FUNCTION_BLOCK CM_SpeedDoor EXTENDS CM_Base IMPLEMENTS I_Door
VAR_INPUT
	i_stSettings : ST_SettingsSpeedDoor;
END_VAR
VAR
	// Inputs
	I_bStaDoorIsOpended AT %I* : BOOL; //Door is opened
	I_bStaDoorIsClosed AT %I* : BOOL; //Door is closed
	I_bStaDoorHasError AT %I* : BOOL; //Door has error
	
	// Outputs
	Q_bCmdOpenDoor AT %Q* : BOOL; //Commnad to open door
	Q_bCmdCloseDoor AT %Q* : BOOL; //Command to close door
	Q_bCmdResetDoor AT %Q* : BOOL; //Command to reset door (controller)
		
	// Requests
	s_bReqClose : BOOL;
	s_bReqOpen : BOOL;
	s_bReqReset : BOOL;
	
	// States
	s_bStaDoorIsClosed : BOOL;
	s_bStaDoorIsClosing : BOOL;
	s_bStaDoorIsOpened : BOOL;
	s_bStaDoorIsOpening : BOOL;
	s_bStaDoorHasError : BOOL;
	
	// Timers
	s_tofResetPulse : TOF;
	s_tonTimeput : TON;
	
	
	// Feedbacks
	arr_sFeedbackName : ARRAY[0..7] OF STRING;
	arr_bFeedbackState : ARRAY[0..7] OF STRING;
	
	
	// Alarms
	s_errSpeedDoor : FB_AlarmHandler;
	s_errTimeout : FB_AlarmHandler;
		
END_VAR


SUPER^();

METHOD PROTECTED _m_Alarms : BOOL
VAR
	nCounter : UDINT;
	
	tTimeout : TIME;
	sMessage : STRING(8);
END_VAR

IF NOT SUPER^._m_Alarms() THEN
	RETURN;
END_IF

s_errSpeedDoor(
	i_bStaActive := i_bReqEnable AND s_bStaDoorHasError, 
	i_eAlarmLevel := E_AlarmLevel.Alarm,
	i_sAlarmText := CONCAT(i_sCmName , CONCAT(': Drive/Controller - ', 'has error (check DYNACO-system)'))
);

IF s_bReqOpen THEN
	tTimeout := i_stSettings.tDoorOpeningTimeout;
	sMessage := 'opening';
ELSIF s_bReqClose THEN
	tTimeout := i_stSettings.tDoorClosingTimeout;
	sMessage :=	'closing';
ELSE
	tTimeout := T#60S;
	sMessage :=	'unknown';	
END_IF
 
s_tonTimeput(
	IN := (s_bReqOpen AND NOT s_bStaDoorIsOpened) OR (s_bReqClose AND NOT s_bStaDoorIsClosed),
	PT := tTimeout
);

s_errTimeout(
	i_bStaActive := i_bReqEnable AND s_tonTimeput.Q, 
	i_eAlarmLevel := E_AlarmLevel.Alarm,
	i_sAlarmText := CONCAT(i_sCmName , CONCAT(': Movement timeout - during ', CONCAT(sMessage, ' (check DYNACO-system)')))
);
	
s_bStaError := s_errSpeedDoor.q_bStaActive OR s_errTimeOut.q_bStaActive;

_m_Alarms := TRUE;
END_METHOD

METHOD PROTECTED _m_Devices : BOOL

VAR
	s_eSeq : E_SeqSpeedDoor;
END_VAR

IF NOT SUPER^._m_Devices() THEN
	RETURN;
END_IF

//Reset request is case of an error
IF s_bStaError THEN
	s_bReqOpen :=
	s_bReqClose := FALSE;
END_IF

CASE s_eSeq OF
	E_SeqSpeedDoor.IDLE:
		;// Some code?
		
	E_SeqSpeedDoor.OPENING:
		;// Some code?
		
	E_SeqSpeedDoor.OPENED:
		;// Some code?
		
	E_SeqSpeedDoor.CLOSING:
		;// Some code?
		
	E_SeqSpeedDoor.CLOSED:
		;// Some code?
		
	E_SeqSpeedDoor.ERROR:
		;// Some code?
		
END_CASE

_m_Devices := TRUE;
END_METHOD

METHOD PROTECTED _m_Hmi : BOOL

IF NOT SUPER^._m_Hmi() THEN
	RETURN;
END_IF

_m_Hmi := TRUE;
END_METHOD

METHOD PROTECTED _m_Init : BOOL

IF NOT SUPER^._m_Init() THEN
	RETURN;
END_IF

{warning '#TODO: Not sure if this control module needs initialzation'}
//--s_DOValve.i_stSettings.bCfgDelay 		:= FALSE;
//--s_DOValve.i_stSettings.tmOutputDelay 	:= T#0S;

_m_Init := TRUE;
END_METHOD

METHOD PROTECTED _m_Inputs : BOOL

IF NOT SUPER^._m_Inputs() THEN
	RETURN;
END_IF

s_bStaDoorIsOpened := I_bStaDoorIsOpended;
s_bStaDoorIsClosed := I_bStaDoorIsClosed;
s_bStaDoorHasError := I_bStaDoorHasError;

_m_Inputs := TRUE;
END_METHOD

METHOD PROTECTED _m_Outputs : BOOL

IF NOT SUPER^._m_Outputs() THEN
	RETURN;
END_IF

s_tofResetPulse(IN := s_bReqReset AND NOT s_tofResetPulse.Q, PT := i_stSettings.tResetPulseDuration);
s_bReqReset := FALSE;
	
Q_bCmdResetDoor := s_tofResetPulse.Q;
Q_bCmdOpenDoor := i_bReqEnable AND s_bReqOpen AND NOT s_bStaDoorIsOpened;
Q_bCmdCloseDoor := i_bReqEnable AND s_bReqClose AND NOT s_bStaDoorIsClosed;
	
_m_Outputs := TRUE;
END_METHOD

METHOD PUBLIC m_Close : BOOL

IF NOT i_bReqEnable THEN 
	RETURN;
END_IF

s_bReqClose := TRUE;
s_bReqOpen := FALSE;
	
m_Close := TRUE;
END_METHOD

METHOD PUBLIC m_Open : BOOL

IF NOT i_bReqEnable THEN 
	RETURN;
END_IF

s_bReqClose := FALSE;
s_bReqOpen := TRUE;
	
m_Open := TRUE;
END_METHOD

METHOD PUBLIC m_Reset : BOOL

IF NOT i_bReqEnable THEN 
	RETURN;
END_IF

s_bReqReset := TRUE;
	
m_Reset := TRUE;
END_METHOD

METHOD PUBLIC m_Stop : BOOL

s_bReqClose := FALSE;
s_bReqOpen := FALSE;
	
m_Stop := TRUE;
END_METHOD

{attribute 'monitoring':='call'}
PROPERTY PUBLIC p_bStaHasError : BOOL
GET

p_bStaHasError := s_bStaError;
END_GET
END_PROPERTY

{attribute 'monitoring':='call'}
PROPERTY PUBLIC p_bStaIsClosed : BOOL
GET

p_bStaIsClosed := s_bStaDoorIsClosed;
END_GET
END_PROPERTY

{attribute 'monitoring':='call'}
PROPERTY PUBLIC p_bStaIsClosing : BOOL
GET

p_bStaIsClosing := s_bReqClose AND NOT s_bStaDoorIsClosed;
END_GET
END_PROPERTY

{attribute 'monitoring':='call'}
PROPERTY PUBLIC p_bStaIsOpened : BOOL
GET

p_bStaIsOpened := s_bStaDoorIsOpened;
END_GET
END_PROPERTY

{attribute 'monitoring':='call'}
PROPERTY PUBLIC p_bStaIsOpening : BOOL
GET

p_bStaIsOpening := s_bReqOpen AND NOT s_bStaDoorIsOpened;
END_GET
END_PROPERTY

END_FUNCTION_BLOCK

(* stored: Version 1.1.0.1, ProductVersion 3.1.4024.12
   POU CM_SpeedDoor: Id {e2ac819d-166f-472e-93dd-5b172f53ac70}, SpecialFunc None
   Folder Methods: Id {dd2ef451-5f00-4ad8-b27b-ac26bc262820}
   Folder Properties: Id {94c06e33-8c98-4e4c-9eed-8612b89d755c}
   Method _m_Alarms: Id {b8083211-2c26-4309-a88e-d066548d2c6f}
   Method _m_Devices: Id {19806151-6bfc-4d1c-84d0-f6d34cd7cf25}
   Method _m_Hmi: Id {7840a539-413d-41f3-9ea8-d8dc0b64e9ee}
   Method _m_Init: Id {ed9edf80-d019-4069-bda1-c3433fdfc559}
   Method _m_Inputs: Id {2072e72c-41a8-4ff9-a497-b847d4491135}
   Method _m_Outputs: Id {b9720cd4-7d4f-42d3-8c4a-83730026236d}
   Method m_Close: Id {7be6b50d-5014-443a-be9d-cc86325ee4dd}
   Method m_Open: Id {49abf2ba-d09f-4bfc-8f29-0007510177f3}
   Method m_Reset: Id {2b94f0b3-4541-4c9a-84a0-3021994a0458}
   Method m_Stop: Id {803f8574-e518-404c-afa9-ff03ca230bc4}
   Property p_bStaHasError: Id {efdb409c-b976-46da-af64-aad420d2e666}
   Get Get: Id {7228a312-914c-416d-9eee-3764a9fb17b5}
   Property p_bStaIsClosed: Id {ef1dc088-110b-467e-86be-7f52cc54884f}
   Get Get: Id {b33ffe41-405f-44dc-9f2a-e98f9f590f06}
   Property p_bStaIsClosing: Id {e38aff16-9321-443b-af16-44540701eeba}
   Get Get: Id {e9c2334a-530d-42a6-9150-7c6498b38b35}
   Property p_bStaIsOpened: Id {32401d29-e49a-4af3-b091-b0c12d3eebf7}
   Get Get: Id {e6852986-45e6-4621-95cd-f7a435ccbaef}
   Property p_bStaIsOpening: Id {8e8ccc3c-3c29-4ab6-808d-63f7f129183c}
   Get Get: Id {03452541-5f72-4a9e-a064-a4ab86d90405} *)
